Staubli VAL3: production.pjx

--- production.pjx ---
Parameters version=s7.5.3 stackSize=5000 millimeterUnit=true
Program file=CycleRefresh.pgx
Program file=getPath.pgx
Program file=loadPage.pgx
Program file=main.pgx
Program file=onEnterEvent.pgx
Program file=onExit.pgx
Program file=onF1Event.pgx
Program file=onF2Event.pgx
Program file=onF3Event.pgx
Program file=onF4Event.pgx
Program file=onF5Event.pgx
Program file=onF6Event.pgx
Program file=onF7Event.pgx
Program file=onF8Event.pgx
Program file=onStart.pgx
Program file=printList.pgx
Program file=printScreen.pgx
Program file=printToShow.pgx
Program file=refresh.pgx
Program file=refreshDynamic.pgx
Program file=refreshPoints.pgx
Program file=refreshProg.pgx
Program file=refreshStatic.pgx
Program file=showLog.pgx
Program file=showMessage.pgx
Program file=simulation.pgx
Data file=production.dtx
Library alias=page path=Disk://kernel/template/page/page.pjx
Library alias=use path=Disk://kernel/userPage/userPage.pjx
Library alias=language path=Disk://kernel/language/language.pjx
Library alias=saveData path=Disk://saveData/saveData.pjx
Library alias=cycleStatus path=Disk://cycleStatus/cycleStatus.pjx
Library alias=usePoint path=Disk://kernel/2/../userPage/userPage.pjx
Library alias=processList path=Disk://kernel/processList/processList.pjx
Library alias=useLog path=Disk://kernel/1/../userPage/userPage.pjx
Library alias=OnEvent path=Disk://OnEvent/OnEvent.pjx
Library alias=saveInputOutput path=Disk://saveInputOutput/saveInputOutput.pjx
Type name=Trajectory path=Disk://kernel/template/Trajectory/Trajectory.pjx
Type name=progItem path=Disk://kernel/template/progItem/progItem.pjx
Type name=dioItem path=Disk://kernel/template/dioItem/dioItem.pjx
Type name=InstrItem path=Disk://kernel/template/InstrItem/InstrItem.pjx

--- production.dtx ---
num nEvent
num nKey = 255
num nMax
num nMin
public num nPage
num nPoint
num nRefresh
num nTime = 5
public num nToSuperV
num nValue
num nIndex
num nSelect
num nView
num nClockScroll
num nFile
string sEvent
public string sItems
string sMenu[4]
  [0] = "HOME"
  [1] = "Emap"
  [2] = "Pallet"
  [3] = "Process"
string sMenu8[8]
string sMessage
string sLogAction
bool bButton[8]
  [0] = true
  [1] = true
  [2] = true
  [3] = true
  [6] = true
bool bLarge
bool bPage
bool bRefreshPoint = true
bool bRefreshProg
bool bShowMessage
bool bTrajLoad
bool bShowInit
bool bUseAutoScroll
num nPointLine[200]
string sProgName
string sTrajName
bool bTraj

--- main.pgx ---
public program main()
  local num i
begin
  // INIT
  if sItems=="simulation"
    call simulation()
  else
    call onStart()
    call refresh()
    // LOOP UNTIL nKey=255
    do
      nKey=getKey()
      switch nKey
        case 259
          //
          //  USE TAB
          //
          bLarge=!bLarge
          cls()
          use:bUseRefresh=true
        break
        case 264,268
          // change from one page to the other one
          bPage=!bPage
          cls()
          use:bUseRefresh=true
        break
        case 271
          call onF1Event()
        break
        case 272
          call onF2Event()
        break
        case 273
          call onF3Event()
        break
        case 274
          call onF4Event()
        break
        case 275
          call onF5Event()
        break
        case 276
          call onF6Event()
        break
        case 277
          call onF7Event()
        break
        case 278
          call onF8Event()
        break
        case 270
          // PAGE PROCESS LIST
          call onEnterEvent()
        break
      endSwitch
      // REFRESH
      call refresh()
      delay(0.1)
    until nKey==255
    // on Exit
    call onExit()
  endIf
end

--- CycleRefresh.pgx ---
program CycleRefresh()
  local string l_sProg
  local num l_nSize[3]
  local num i
  local num l_nResult
  local num l_nPointView
  local Trajectory l_tTraj
begin
  // set SIZE LIST
  if !bLarge
    // one HALF right
    call use:setSizeList(19,0,19,10)
  elseIf cycleStatus:bTraj
    // one HALF LEFT
    call use:setSizeList(0,0,18,10)
  else
    // FULL
    call use:setSizeList(0,0,38,10)
  endIf
  // POINT LIST
  call usePoint:setSizeList(19,0,19,10)
  // check the update
  if bTraj!=cycleStatus:bTraj
    bTraj=cycleStatus:bTraj
    use:bUseRefresh=true
  endIf
  // PROGRAM
  if use:bUseRefresh or(sProgName!=cycleStatus:pCycleProg.sID)
    // get the name
    sProgName=cycleStatus:pCycleProg.sID
    // build the program list and build the list
    call printScreen()
    call refreshProg(cycleStatus:pCycleProg)
    // show the list
    nEvent=cycleStatus:nEvent
    use:nView=nEvent%use:nBottomY
    call use:listupdate(nEvent-use:nView)
    bRefreshPoint=true
    // CHECK THE LINE NUMBER
  elseIf nEvent!=cycleStatus:nEvent
    nEvent=cycleStatus:nEvent
    if use:nView>=nEvent%use:nBottomY
      // refresh the list
      use:nView=nEvent%use:nBottomY
      call use:listupdate(nEvent-use:nView)
    else
      // just the line
      call use:listcursor(use:nView,false)
      call use:listcursor(nEvent%use:nBottomY,true)
    endIf
  endIf
  // TRAJECTORY
  if cycleStatus:bTraj
    // get the first trajectory
    call cycleStatus:getTraj(l_tTraj)
    if l_tTraj.sID!="null" and l_tTraj.sID!=""
      if use:bUseRefresh or bRefreshPoint or sTrajName!=l_tTraj.sID
        //
        // rebuilt the Traj list
        //
        call refreshPoints(l_tTraj)
        nPoint=cycleStatus:nPoint
        l_nPointView=nPointLine[nPoint]
        usePoint:nView=l_nPointView%usePoint:nBottomY
        //        if bRefreshPoint
        //          bRefreshPoint=false
        //          call usePoint:listupdate(l_nPointView-usePoint:nView)
        //        else
        call usePoint:listupdate(l_nPointView-usePoint:nView)
        //        endIf
      else
        // just the line
        if nPoint!=cycleStatus:nPoint
          nPoint=cycleStatus:nPoint
          l_nPointView=nPointLine[nPoint]
          if usePoint:nView>=l_nPointView%usePoint:nBottomY
            // update the list
            usePoint:nView=l_nPointView%usePoint:nBottomY
            call usePoint:listupdate(l_nPointView-usePoint:nView)
          else
            //just the line
            call usePoint:listcursor(usePoint:nView,false)
            usePoint:nView=l_nPointView%usePoint:nBottomY
            call usePoint:listcursor(usePoint:nView,true)
          endIf
        endIf
      endIf
    endIf
  endIf
end

--- getPath.pgx ---
program getPath(string& x_sType[] (dimensions=1))
  local num l_nPos
  local string l_sPath
begin
  // get the TypePath
  l_sPath=x_sType
  do
    l_nPos=find(l_sPath,"/")
    if l_nPos==-1
      l_nPos=find(l_sPath,"\")
    endIf
    if l_nPos!=-1
      l_sPath=right(l_sPath,len(l_sPath)-l_nPos-1)
    endIf
  until l_nPos==-1
  x_sType=l_sPath
end

--- loadPage.pgx ---
program loadPage(string x_sPage, string& x_sItems[])
// load the next page
  local num i
  local string l_sMessage
begin
  // look if the page libload is correct
  i=page:libLoad(x_sPage)
  delay(0)
  if i!=0
    logMsg("[KERNEL] INTERFACE:PAGE LIBLOAD "+x_sPage+" result "+toString("",i))
    call language:message(l_sMessage,-7)
    popUpMsg(l_sMessage+x_sPage+" ; "+toString("",i))
  else
    // copy all the field from x_sItems to the next page
    call use:stringCopy(x_sItems,page:sItems)
    call page:main()
    // to give back
    call use:stringCopy(page:sItems,x_sItems)
    //
    bShowMessage=false
    use:bUseRefresh=true
  endIf
end

--- onEnterEvent.pgx ---
program onEnterEvent()
  local num l_nResult
  local string l_sMessage
  local string l_sMessage2
  local string l_sMessage3
  local string l_sItem
begin
  //if saveData:mode>0
  if !bPage
    //
    //  open the processes list PAGE
    //
    //      saveData:sProcessList="default"
    //      call processList:loadProcessList(saveData:sProcessList,l_nResult)
    l_sItem="true"
    call loadPage("kernel/page/processList",l_sItem)
    // came back
    logMsg("[KERNEL] INTERFACE:PAGE Production")
    // refresh
    cls()
    use:bUseRefresh=true
  endIf
  //endIf
end

--- onExit.pgx ---
program onExit()
begin
  //
end

--- onF1Event.pgx ---
program onF1Event()
  local num l_nValue[4]
  local string l_sItem[4]
  local string l_sMessage
  local num l_nMin[4]
  local num l_nMax[4]
  local bool l_bLarge
  local num l_nKey
begin
  // look if the bButton is enable
  if bButton[0]
    //
    if !bPage
      // normal production page
      if cycleStatus:bCycle==false
        //and cycleStatus:bIsHome==false
        //
        if cycleStatus:nWorkingMode==1
          if isPowered()==false
            call language:message(l_sMessage,201)
            call use:timerDialog(l_sMessage,0)
            do
              l_nKey=getKey()
              if l_nKey==255 or cycleStatus:nWorkingMode!=1
                return
              endIf
              delay(0)
            until isPowered()
          endIf
          l_bLarge=bLarge
          cls()
          cycleStatus:bToHome=true
          wait(cycleStatus:bToHome==false)
          call simulation()
          //
          bLarge=l_bLarge
        else
          call language:message(l_sMessage,92)
          call use:timerDialog(l_sMessage,2)
        endIf
      endIf
    else
      // export the file
      call language:message(l_sMessage,96)
      l_sMessage=l_sMessage+":# actionLog.txt file"
      call use:timerDialog(l_sMessage,0)
      nFile=$fileOpen("actionLog.txt","w")
      $fileSet(nFile,cycleStatus:sLog,size(cycleStatus:sLog))
      $fileClose(nFile)
    endIf
  endIf
end

--- onF2Event.pgx ---
program onF2Event()
begin
  // look if the bButton is enable
  if bButton[1]
    //
  endIf
end

--- onF3Event.pgx ---
program onF3Event()
  local string l_sEmpty
begin
  // look if the bButton is enable
  if bButton[2]
    // load the page Pallet
    l_sEmpty=""
    call loadPage("trajectory/PALLET/page_viewPallet",l_sEmpty)
  endIf
end

--- onF4Event.pgx ---
program onF4Event()
begin
  // look if the bButton is enable
  if bButton[3]
    //

  endIf
end

--- onF5Event.pgx ---
program onF5Event()
begin
  // look if the bButton is enable
  if bButton[4]
    //
    // on F5 button
    //
  endIf
end

--- onF6Event.pgx ---
program onF6Event()
begin
  // look if the bButton is enable
  if bButton[5]
    //
    // PAUSE / RESUME
    //
    if !cycleStatus:bPause
      logMsg("[KERNEL] INTERFACE:Pause cycle")
      call OnEvent:pauseCycle()
    else
      logMsg("[KERNEL] INTERFACE:Resume cycle")
      call OnEvent:resumeCycle()
    endIf
  endIf
end

--- onF7Event.pgx ---
program onF7Event()
  local string l_sMessage
  local bool l_bContinue
  local string l_sProgram
  local num l_nZero
begin
  // look if the bButton is enable
  if bButton[6]
    //
    // STOP/START CYCLE
    //
    if cycleStatus:bCycle
      logMsg("[KERNEL] INTERFACE:Stop cycle")
      stopMove()
      cycleStatus:bToStop=true
      call use:timerDialog(" STOP CYCLE ",1)
      watch(cycleStatus:bToStop==false,1)
    else
      // start cycle
      l_nZero=0
      call processList:getCycle(l_sProgram,l_nZero,l_nZero,l_nZero,1)
      if l_sProgram!=""
        //if (cycleStatus:nWorkingMode==3 or cycleStatus:nWorkingMode==4)
        logMsg("[KERNEL] INTERFACE:Start cycle")
        cycleStatus:bToStart=true
        wait(cycleStatus:bToStart==false)
      else
        // program in the process List
        call language:message(l_sMessage,91)
        popUpMsg(l_sMessage)
      endIf
    endIf
    call use:nullKey(nKey)
  endIf
end

--- onF8Event.pgx ---
program onF8Event()
  local string l_sMessage
begin
  // look if the bButton is enable
  if bButton[7]
    //
    //
    // TERMINATE CYCLE
    //
    if cycleStatus:bCycle and !cycleStatus:bEnding
      logMsg("[KERNEL] INTERFACE:End cycle")
      //
      cycleStatus:bToEnd=true
      call language:message(l_sMessage,3)
      popUpMsg(l_sMessage)
    endIf
  endIf
end

--- onStart.pgx ---
program onStart()
  local num i
  local string l_sPath
begin
  // define the page
  cls()
  // set small wiew
  bLarge=false
  bPage=false
  bShowInit=false
  // INIT the resource
  use:bUseRefresh=true
  logMsg("[KERNEL] INTERFACE:PAGE Production")
end

--- printList.pgx ---
program printList(num x_nType (dimensions=1))
  local num i
  local num l_nX
  local string l_sProg
  local num l_nIndex
  local num l_nSize[3]
  local num l_nDone
  local num l_nTotal
  local num l_nZero
begin
  //
  l_nZero=0
  call use:getListPosition(l_nX,l_nZero)
  // get the size
  call processList:getSize(l_nSize,x_nType)
  // resize it
  if l_nSize!=0
    l_nSize=l_nSize-1
  endIf
  // print the process start LIST
  for i=cycleStatus:nProg to min(l_nSize-cycleStatus:nProg,1)
    call processList:getCycle(l_sProg,l_nTotal,l_nDone,i,x_nType)
    if l_sProg!=""
      if i==cycleStatus:nProg
        setTextMode(1)
      endIf
      call use:strfill(l_sProg,10,l_sProg)
      l_sProg=l_sProg+"["+toString("1",l_nDone)+"/"+toString("1",l_nTotal)+"]"
      call use:type(0,i+1,l_sProg)
      setTextMode(0)
      call use:typeLen(len(l_sProg),i+1,"",l_nX-1-len(l_sProg))
      l_nIndex=l_nIndex+1
    endIf
  endFor
  // write the empty space
  if l_nIndex<2
    for i=l_nIndex to 1
      // empty Line
      call use:typeLen(0,i+1,"",l_nX-1)
    endFor
  endIf
end

--- printScreen.pgx ---
program printScreen()
begin
  if bLarge and bTraj
    // print the screen... easy way
    gotoxy(0,0)
    //     0123456789012345678901234567890123456789
    putln("┌   ───────────────┌   ────────────────┐")
    putln("│                  │")
    putln("│                  │")
    putln("│                  │")
    putln("│                  │")
    putln("│                  │")
    putln("│                  │")
    putln("│                  │")
    putln("│                  │")
    putln("│                  │")
    putln("│                  │")
    putln("└──────────────────")
  elseIf bLarge
    gotoxy(0,0)
    putln("┌   ───────────────────────────────────┐")
    putln("│                                      │")
    putln("│                                      │")
    putln("│                                      │")
    putln("│                                      │")
    putln("│                                      │")
    putln("│                                      │")
    putln("│                                      │")
    putln("│                                      │")
    putln("│                                      │")
    putln("│                                      │")
    putln("└──────────────────────────────────────┘")
  elseIf !bLarge
    // print the screen... easy way
    gotoxy(19,0)
    //    0123456789012345678901234567890123456789
    putln("┌   ────────────────┐")
    gotoxy(19,1)
    putln("│                   │")
    gotoxy(19,2)
    putln("│                   │")
    gotoxy(19,3)
    putln("│                   │")
    gotoxy(19,4)
    putln("│                   │")
    gotoxy(19,5)
    putln("│                   │")
    gotoxy(19,6)
    putln("│                   │")
    gotoxy(19,7)
    putln("│                   │")
    gotoxy(19,8)
    putln("│                   │")
    gotoxy(19,9)
    putln("│                   │")
    gotoxy(19,10)
    putln("│                   │")
    gotoxy(19,11)
    putln("└───────────────────┘")
  endIf
end

--- printToShow.pgx ---
program printToShow()
  local string l_sMessage
  local num i
begin
  //
  //  Print the instruction
  //
  if !bPage
    call use:typeLen(0,12,cycleStatus:sToShow,40)
  endIf
  // print the bar
  if !cycleStatus:bSimulation
    //
    //
    // set the view of the page..
    //
    // SET THE PAGE NUMBER
    use:nPage=20
    // USE <>PROFILE for <>PAGE
    use:nPage=use:nPage+abs(limit(saveData:mode,0,2)-2)
    if cycleStatus:bCycle
      use:nPage=use:nPage+3
    endIf
    // load the menu page
    if saveData:language!="japanese"
      // SET THE VIEW OF THE PAGE
      call language:page(l_sMessage,use:nPage)
      // define the menu
      call use:stringToArray(l_sMessage,sMenu)
    else
      // japanese use the array for the menu
      call language:page(sMenu8,use:nPage)
      call use:stringCopy(sMenu8,sMenu)
    endIf
    // set the HOME button as no button if not need
    if cycleStatus:bCycle or cycleStatus:bIsHome
      sMenu[0]=""
    endIf
    // if the action list is show do not use the first 4 button
    if bPage
      for i=0 to size(sMenu)-1
        sMenu[i]=""
      endFor
      sMenu="Export"
    endIf
    call use:setMenu(sMenu,true,-1)
    call use:getMenu(sMenu,bButton)
    //
    // print to video the Process List-Pause-END-STOP
    //
    // START END
    bButton[6]=true
    if !cycleStatus:bCycle
      if cycleStatus:bIsHome or saveData:bNoUseHome
        call use:type(31,13,"START")
        bButton[6]=true
      endIf
    else
      bButton[5]=true
      // PAUSE
      if !cycleStatus:bPause
        call use:type(24,13,"  PAUSE")
      else
        call use:type(24,13,"RESTART")
      endIf
      call use:type(31,13," STOP ")
      bButton[6]=true
    endIf
    if cycleStatus:bCycle and !cycleStatus:bEnding
      bButton[7]=true
      call use:type(37,13,"END")
    else
      bButton[7]=false
      call use:type(37,13,"   ")
    endIf
  endIf
  // show the trajectory status
  if cycleStatus:bTraj and !bPage
    // show the trajectory status
    call usePoint:scroll(usePoint:nBottomX,usePoint:nBottomY+1,40-usePoint:nBottomX-2,cycleStatus:nIdPercentage)
  endIf
  //
end

--- refresh.pgx ---
program refresh()
// // page refresh
  local string l_sMessage
begin
  // check the page
  if !bPage
    if !bShowMessage
      if (nKey>=270 and nKey<=278)or abs(clock()-nRefresh)>nTime or use:bUseRefresh
        if (nKey>=270 and nKey<=278)or use:bUseRefresh
          cls()
        endIf
        // refresh the static message
        use:bUseRefresh=true
        call refreshStatic()
        call refreshDynamic()
        // update the clock
        nRefresh=clock()
      else
        // refresh the Dynamic message
        call refreshDynamic()
      endIf
    endIf
    // print the message
    call showMessage()
  else
    call showLog()
  endIf
  call printToShow()
end

--- refreshDynamic.pgx ---
program refreshDynamic()
begin
  // DO NOT CHANGE
  //
  // ADD HERE
  //
  call CycleRefresh()
  // print the instruction and the bar
  call printToShow()
  //
  // init
  use:bUseRefresh=false
  //
  // ADD HERE
  //
end

--- refreshPoints.pgx ---
program refreshPoints(Trajectory& x_tTraj[])
  local num i
  local num l_nSize
  local string l_sEvent
  local string l_sItem
  local num j
  local num l_nIndex
  local string l_sData
  local string l_sType
begin
  // create the list
  call usePoint:type(21,0,x_tTraj.sID)
  // get the size
  call usePoint:listempty()
  l_nSize=size(x_tTraj.tSuper)
  for i=0 to l_nSize-1
    // add..
    l_sEvent=x_tTraj.tSuper[i].comment
    l_sItem=toString("2",i+1)+" "+l_sEvent
    nPointLine[i]=l_nIndex
    call usePoint:listadd(l_sItem)
    l_nIndex=l_nIndex+1
    if saveData:bShowItem
      // search for tCP ON OFF
      if x_tTraj.tSuper[i].nTcpAction==1
        l_sItem="  -TCP ON"
      elseIf x_tTraj.tSuper[i].nTcpAction==2
        l_sItem="  -TCP OFF"
      endIf
      if x_tTraj.tSuper[i].nTcpAction>0
        call usePoint:listadd(l_sItem)
        l_nIndex=l_nIndex+1
      endIf
      // scan the action...
      for j=0 to size(x_tTraj.tSuper[i].iInstr)-1
        if x_tTraj.tSuper[i].iInstr[j].sType!=""
          l_sData=x_tTraj.tSuper[i].iInstr[j].sData
          l_sType=x_tTraj.tSuper[i].iInstr[j].sType
          call saveInputOutput:replaceIO(l_sData,l_sType,l_sData)
          l_sItem=l_sType+" "+l_sData
          l_sItem="  -"+l_sItem
          call usePoint:listadd(l_sItem)
          l_nIndex=l_nIndex+1
        endIf
      endFor
    endIf
  endFor
end

--- refreshProg.pgx ---
program refreshProg(progItem& x_pProg[])
  local num i
  local num l_nSize
  local string l_sEvent
  local string l_sTitle
  local progItem l_pProg
  local string l_sData
begin
  // set the size of the windows
  if !(cycleStatus:bTraj)
    call use:setView(bLarge)
  endIf
  // Create the list
  if bLarge
    call use:type(2,0,sProgName)
  else
    call use:type(21,0,sProgName)
  endIf
  // fill IT
  call use:listempty()
  if sProgName!=""
    l_nSize=size(x_pProg.iEvent)
    for i=0 to l_nSize-1
      l_nSize=size(x_pProg.iEvent)
      // insert all
      if i<=size(x_pProg.iEvent)-1
        l_sData=x_pProg.iEvent[min(i,size(x_pProg.iEvent)-1)].sData
        l_sEvent=x_pProg.iEvent[min(i,size(x_pProg.iEvent)-1)].sType
        call saveInputOutput:replaceIO(l_sData,l_sEvent,l_sData)
        l_sEvent=l_sEvent+" "+l_sData
        l_sEvent=toString("2",i+1)+" "+l_sEvent
        call use:listadd(l_sEvent)
      else
        return
      endIf
    endFor
  endIf
end

--- refreshStatic.pgx ---
program refreshStatic()
  local string l_sMenu
  local string l_sMessage
  local num l_nPreset
  local num i
  local num l_nX
  local num l_nProcessType
  local bool l_bMode
  local string l_sProgram
  local num l_nY
  local num l_nZero
begin
  // clear the button line
  call use:clear(0,13)
  //
  // print to video info of all
  //
  if !bLarge
    call use:getListPosition(l_nX,l_nY)
    // line 0
    call use:typeLen(0,0,"",l_nX-1)
    // line 1-2
    //
    // print to video the first 2 program in the process List
    //
    l_nProcessType=cycleStatus:nProcessType
    // show the nProcessTypeis the start List empty
    l_nZero=0
    call processList:getCycle(l_sProgram,l_nZero,l_nZero,l_nZero,0)
    if l_sProgram=="" and l_nProcessType==0
      l_nProcessType=1
    endIf
    // PRINT THE PROGRAM LIST
    call printList(l_nProcessType)
    // line 3
    //  print to video the clock
    call language:message(l_sMessage,90)
    call use:strfill(l_sMessage+" "+toString(".2",cycleStatus:nCycleTime),use:nBottomX,l_sMessage)
    call use:typeLen(0,3,"",l_nX-1)
    call use:typeLen(0,4,l_sMessage,l_nX-1)
    // line 4
    call use:typeLen(0,5,"",l_nX-1)
    //line 5
    l_sMessage=""
    call use:typeLen(0,6,l_sMessage,l_nX-1)
    // line 7- 11 none
    for i=7 to 11
      call use:typeLen(0,i," ",l_nX-1)
    endFor
  endIf
  // check the if the robot is at home
  call language:message(l_sMessage,223)
  if !cycleStatus:bIsHome and !cycleStatus:bCycle and !cycleStatus:bSimulation
    // ROBOT IS NOT AT HOME
    cycleStatus:sToShow=l_sMessage
    // reset the signal
  elseIf cycleStatus:sToShow==l_sMessage
    cycleStatus:sToShow=""
  endIf
end

--- showLog.pgx ---
program showLog()
  local num l_nSize
  local num i
begin
  // show the log items
  setMutex(cycleStatus:bMutex)
  // check the size
  if size(cycleStatus:sLog)<size(useLog:sItems) or bShowInit==false
    // create the list
    call useLog:setSizeList(0,0,38,11)
    call useLog:listcreate("action log")
    nSelect=-1
    bShowInit=true
  elseIf use:bUseRefresh
    // refresh the list
    call useLog:listredraw(size(useLog:sItems))
    use:bUseRefresh=false
  endIf
  // check if need to add value
  l_nSize=sel(cycleStatus:sLog=="",0,size(cycleStatus:sLog))-sel(useLog:sItems=="",0,size(useLog:sItems))
  if l_nSize!=0
    // add the items
    call useLog:listadd(cycleStatus:sLog[size(cycleStatus:sLog)-l_nSize])
  endIf
  //release
  cycleStatus:bMutex=false
  // refresh
  // update the scrooling
  call useLog:selectNewField(nSelect,nIndex,nView)
  call useLog:listevent(nKey,nIndex,sLogAction)
  // wait 5 sec
  if nKey==-1 and clock()-nClockScroll>5
    bUseAutoScroll=true
  elseIf nKey!=-1
    bUseAutoScroll=false
    nClockScroll=clock()
  endIf
  if bUseAutoScroll
    // update to the last item
    nSelect=size(cycleStatus:sLog)-1
  else
    nSelect=nIndex
  endIf
  // update
  nView=useLog:nView
end

--- showMessage.pgx ---
program showMessage()
  local string l_sMessage
  local string l_sMessage2
  local bool l_bTollerance
begin
  // INIT
  bShowMessage=false
  // look for the esStatus
  if esStatus()==2
    call language:message(l_sMessage,222)
  elseIf cycleStatus:bCycle or cycleStatus:bSimulation
    //
    // PRIORITY
    //
    // 1) GO TO MANUAL IF OUTSIDE JOINT SECURE ZONE
    // 2) GO TO AUTO MODE OR PRESS RESTART
    // 3) CONNECTION MOVE
    // 4) PRESS RESTART
    // 5) POWER ON
    // 6) PRESS MOVE HOLD
    // 7) JOINT / WORLD / TOOL
    // check the tollerance
    call cycleStatus:checkTollerance(l_bTollerance)
    //
    if !l_bTollerance and (cycleStatus:nWorkingMode==4 or cycleStatus:nWorkingMode==3) and cycleStatus:bPause
      // ASK to GO manual to continue the connection movement
      call language:message(l_sMessage,92)
      call language:message(l_sMessage2,145)
      l_sMessage=l_sMessage+"#"+l_sMessage2
    elseIf l_bTollerance and cycleStatus:nWorkingMode==1 and cycleStatus:bPause
      // ASK TO GO TO AUTO MODE AND PRESS RESTART
      call language:message(l_sMessage,200)
      call language:message(l_sMessage2,144)
      l_sMessage=l_sMessage+"#"+l_sMessage2
    elseIf cycleStatus:nWorkingStatus==1 and cycleStatus:nWorkingMode!=3 and cycleStatus:nWorkingMode!=4 and isPowered() and cycleStatus:bPause
      // connection movement
      call language:message(l_sMessage,145)
    elseIf cycleStatus:bPause and l_bTollerance
      //and(cycleStatus:nWorkingMode==3 or cycleStatus:nWorkingMode==4)
      // press restart to continue
      call language:message(l_sMessage,144)
    elseIf (cycleStatus:nWorkingMode!=4 and !isPowered())
      // POWER ON
      call language:message(l_sMessage,201)
    elseIf cycleStatus:nWorkingMode==4 and cycleStatus:nWorkingStatus==2 and !isPowered()
      // settling the power...
      call language:message(l_sMessage,146)
      call use:timerDialog(l_sMessage,0.2)
      if watch(cycleStatus:nWorkingStatus!=2,2)
        // exit
        return
      endIf
    elseIf (cycleStatus:nWorkingStatus!=0)
      if isEmpty()
        // PRESS MOVE HOLD
        call language:message(l_sMessage,130)
      else
        // PRESS MOVE HOLD
        call language:message(l_sMessage,203)
      endIf
      // MANUAL MODE
      if cycleStatus:nWorkingMode==1
        switch cycleStatus:nWorkingStatus
          case 2
            // JOINT
            call language:message(l_sMessage,140)
          break
          case 3
            // WORLD
            call language:message(l_sMessage,141)
          break
          case 4
            // TOOL
            call language:message(l_sMessage,142)
          break
          case 5
            // POINT
            call language:message(l_sMessage,143)
          break
        endSwitch
      endIf
    endIf
  endIf
  // show message
  if l_sMessage!=""
    bShowMessage=true
    call use:timerDialog(l_sMessage,0.1)
  endIf
end

--- simulation.pgx ---
program simulation()
  local string l_sMessage
begin
  //
  // SIMULATION
  //
  // syncro
  bLarge=true
  use:nPage=200
  watch(cycleStatus:pCycleProg.sID!="",1)
  use:bUseRefresh=true
  cls()
  do
    nKey=getKey()
    // REFRESH
    if cycleStatus:bSimulation
      call refresh()
    endIf
    call use:type(31,13,"STOP ")
    // look for the restart button
    if cycleStatus:bPause
      call use:type(23,13,"RESTART")
      if nKey==276
        call OnEvent:resumeCycle()
      endIf
    else
      call use:type(23,13,"        ")
    endIf
    delay(0)
  until nKey==255 or nKey==277 or cycleStatus:bToStop or cycleStatus:bSimulation==false
  //
  if nKey==255 or nKey==277
    cycleStatus:bToStop=true
    watch(cycleStatus:bToStop==false,1)
  endIf
  // leave
  call use:nullKey(nKey)
end
